// Mitsubishi GX Works2 project: MixerDUrcpp8pumps   PLC: FX3U/FX3UC

PROGRAM MAIN
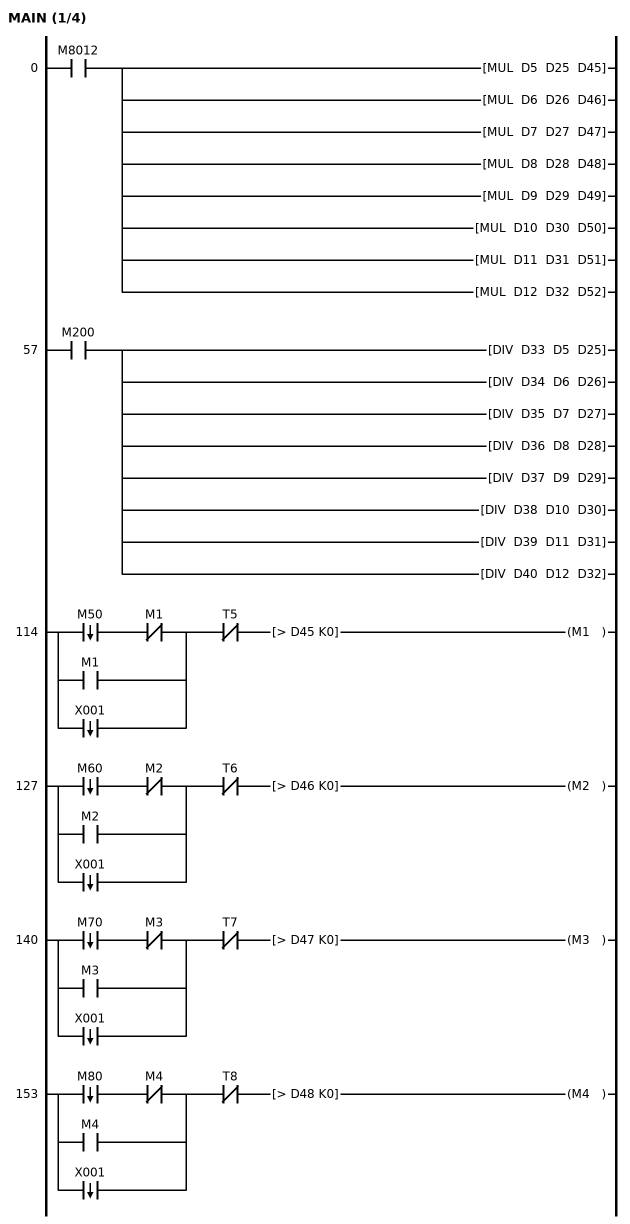
0     LD      M8012
      MUL     D5 D25 D45
      MUL     D6 D26 D46
      MUL     D7 D27 D47
      MUL     D8 D28 D48
      MUL     D9 D29 D49
      MUL     D10 D30 D50
      MUL     D11 D31 D51
      MUL     D12 D32 D52
57    LD      M200
      DIV     D33 D5 D25
      DIV     D34 D6 D26
      DIV     D35 D7 D27
      DIV     D36 D8 D28
      DIV     D37 D9 D29
      DIV     D38 D10 D30
      DIV     D39 D11 D31
      DIV     D40 D12 D32
114   LDF     M50
      ANI     M1
      OR      M1
      ORF     X001
      ANI     T5
      AND>    D45 K0
      OUT     M1
127   LDF     M60
      ANI     M2
      OR      M2
      ORF     X001
      ANI     T6
      AND>    D46 K0
      OUT     M2
140   LDF     M70
      ANI     M3
      OR      M3
      ORF     X001
      ANI     T7
      AND>    D47 K0
      OUT     M3
153   LDF     M80
      ANI     M4
      OR      M4
      ORF     X001
      ANI     T8
      AND>    D48 K0
      OUT     M4
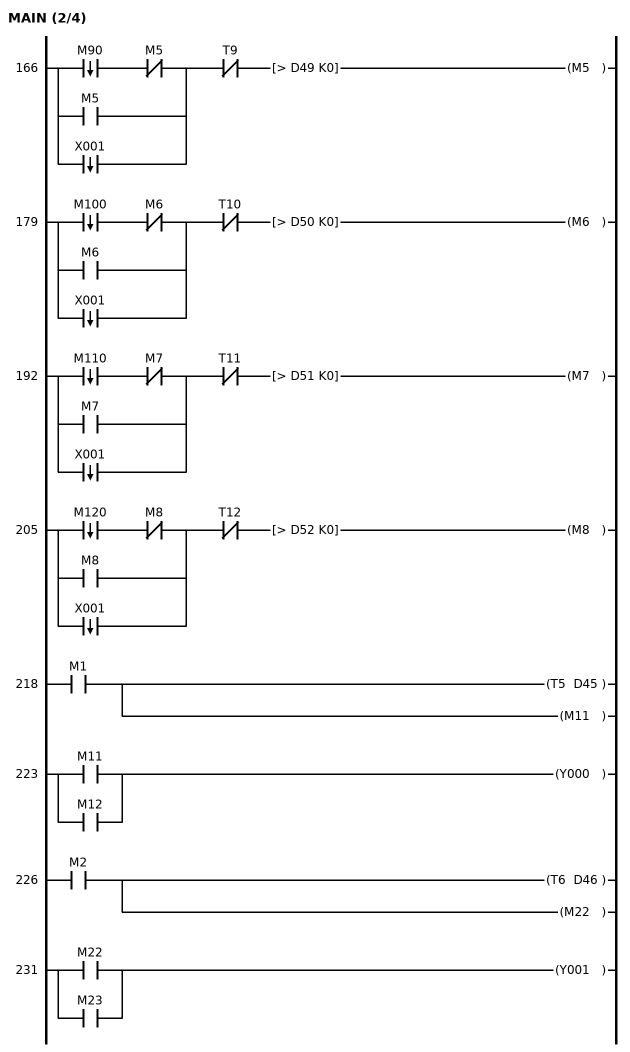
166   LDF     M90
      ANI     M5
      OR      M5
      ORF     X001
      ANI     T9
      AND>    D49 K0
      OUT     M5
179   LDF     M100
      ANI     M6
      OR      M6
      ORF     X001
      ANI     T10
      AND>    D50 K0
      OUT     M6
192   LDF     M110
      ANI     M7
      OR      M7
      ORF     X001
      ANI     T11
      AND>    D51 K0
      OUT     M7
205   LDF     M120
      ANI     M8
      OR      M8
      ORF     X001
      ANI     T12
      AND>    D52 K0
      OUT     M8
218   LD      M1
      OUT     T5 D45
      OUT     M11
223   LD      M11
      OR      M12
      OUT     Y000
226   LD      M2
      OUT     T6 D46
      OUT     M22
231   LD      M22
      OR      M23
      OUT     Y001
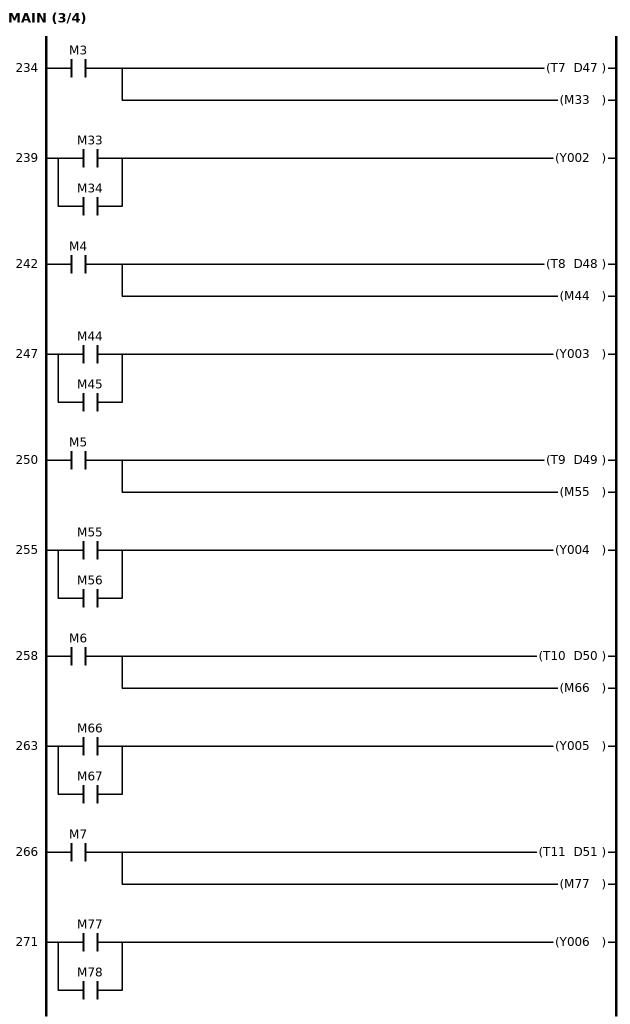
234   LD      M3
      OUT     T7 D47
      OUT     M33
239   LD      M33
      OR      M34
      OUT     Y002
242   LD      M4
      OUT     T8 D48
      OUT     M44
247   LD      M44
      OR      M45
      OUT     Y003
250   LD      M5
      OUT     T9 D49
      OUT     M55
255   LD      M55
      OR      M56
      OUT     Y004
258   LD      M6
      OUT     T10 D50
      OUT     M66
263   LD      M66
      OR      M67
      OUT     Y005
266   LD      M7
      OUT     T11 D51
      OUT     M77
271   LD      M77
      OR      M78
      OUT     Y006
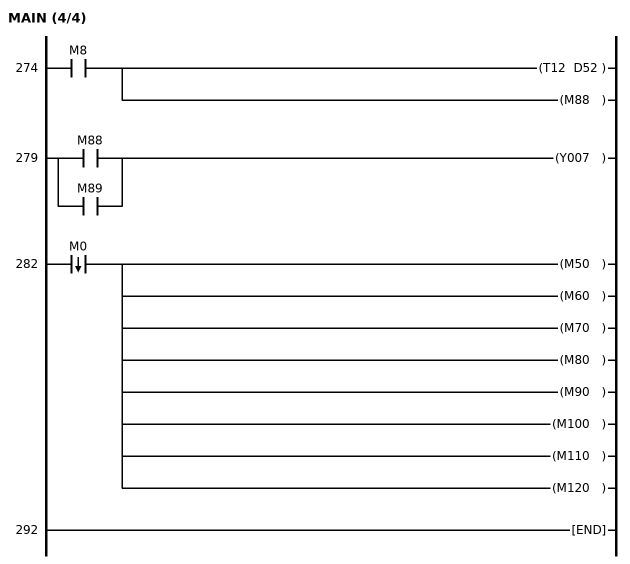
274   LD      M8
      OUT     T12 D52
      OUT     M88
279   LD      M88
      OR      M89
      OUT     Y007
282   LDF     M0
      OUT     M50
      OUT     M60
      OUT     M70
      OUT     M80
      OUT     M90
      OUT     M100
      OUT     M110
      OUT     M120
292   END
END_PROGRAM
